SUBAPPLICATION Uebung_134 (* Übung zu ISOBUS Receive from Unclaimed Partner *)
  (* Standard: 61499-2; Description: Copyright (c) 2026 Meisterschulen am Ostbahnhof This program and the accompanying materials are made available under the terms of the Eclipse Public License 2.0 which is available at https://www.eclipse.org/legal/epl-2.0/ SPDX-License-Identifier: EPL-2.0 *)
  (* Version 1.0, 2026-01-16, Gemini, Meisterschulen am Ostbahnhof *)
  PACKAGE Uebungen;
  IMPORT Uebungen::const::Uebung_120_129::Filter::FLT_ALL_PASS;
  IMPORT isobus::pgn::ISOUSERHOME_e::thisMember;
  IMPORT isobus::pgn::ISO_CAN_NODE::NODE1;
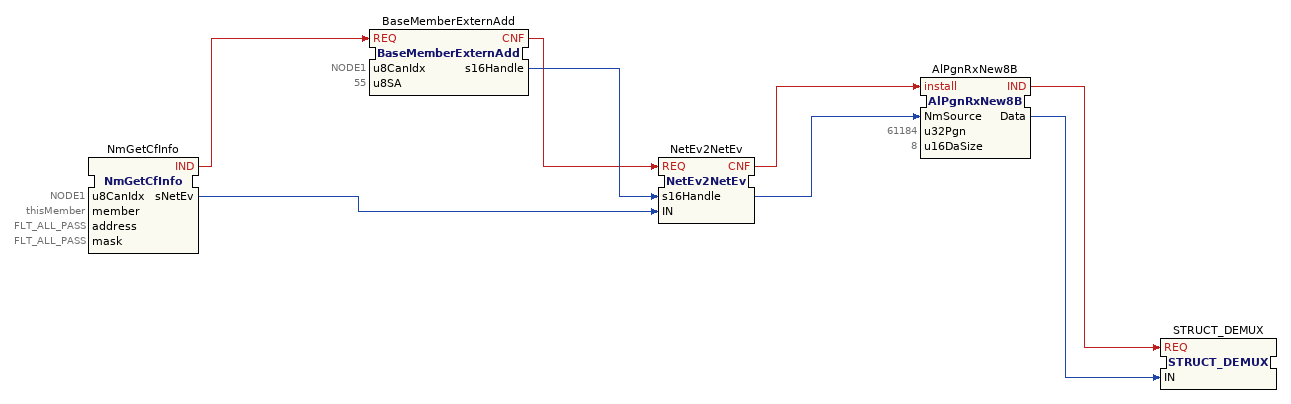
  FBS
    BaseMemberExternAdd : isobus::pgn::BaseMemberExternAdd(u8CanIdx := NODE1, u8SA := 55);
    AlPgnRxNew8B : isobus::pgn::rx::AlPgnRxNew8B(u32Pgn := 61184, u16DaSize := 8);
    NmGetCfInfo : isobus::pgn::NmGetCfInfo(u8CanIdx := NODE1, member := thisMember, address := FLT_ALL_PASS, mask := FLT_ALL_PASS);
    NetEv2NetEv : isobus::pgn::NetEv2NetEv;
    STRUCT_DEMUX : eclipse4diac::convert::STRUCT_DEMUX; {SET_ATTRIBUTE(StructuredType, isobus::pgn::CAN_MSG)}
  END_FBS
  EVENT_CONNECTIONS
    BaseMemberExternAdd.CNF TO NetEv2NetEv.REQ;
    NetEv2NetEv.CNF TO AlPgnRxNew8B.install;
    NmGetCfInfo.IND TO BaseMemberExternAdd.REQ;
    AlPgnRxNew8B.IND TO STRUCT_DEMUX.REQ;
  END_CONNECTIONS
  DATA_CONNECTIONS
    BaseMemberExternAdd.s16Handle TO NetEv2NetEv.s16Handle;
    NmGetCfInfo.sNetEv TO NetEv2NetEv.IN;
    NetEv2NetEv. TO AlPgnRxNew8B.NmSource;
    AlPgnRxNew8B.Data TO STRUCT_DEMUX.IN;
  END_CONNECTIONS
END_SUBAPPLICATION
